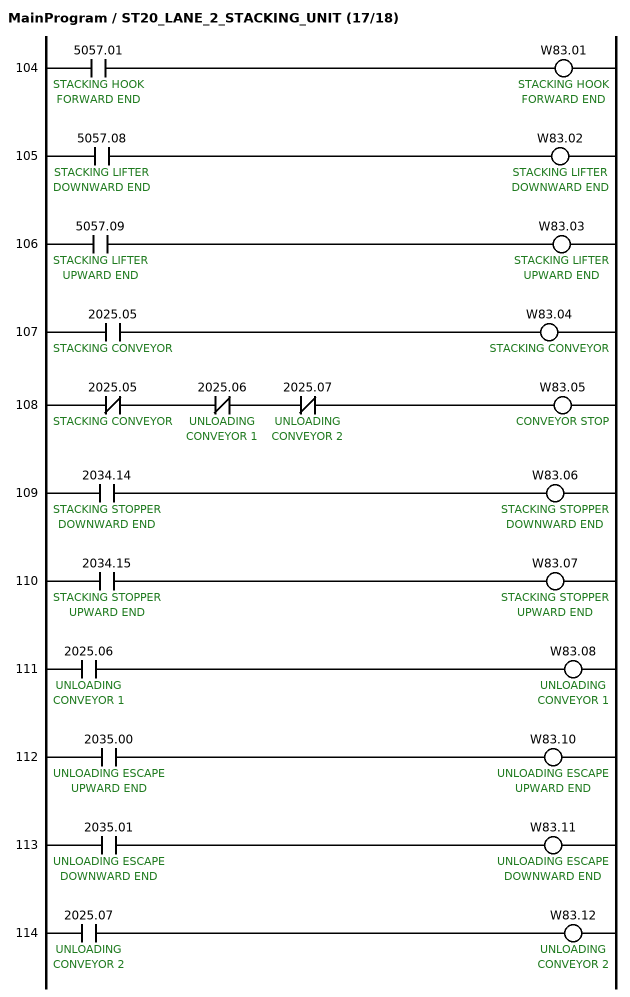
; [picture p720: MainProgram / ST20_LANE_2_STACKING_UNIT, rungs 104-114]
; rung 104
LD 5057.01  ; STACKING HOOK FORWARD END
OUT W83.01  ; STACKING HOOK FORWARD END
; rung 105
LD 5057.08  ; STACKING LIFTER DOWNWARD END
OUT W83.02  ; STACKING LIFTER DOWNWARD END
; rung 106
LD 5057.09  ; STACKING LIFTER UPWARD END
OUT W83.03  ; STACKING LIFTER UPWARD END
; rung 107
LD 2025.05  ; STACKING CONVEYOR
OUT W83.04  ; STACKING CONVEYOR
; rung 108
LDNOT 2025.05  ; STACKING CONVEYOR
ANDNOT 2025.06  ; UNLOADING CONVEYOR 1
ANDNOT 2025.07  ; UNLOADING CONVEYOR 2
OUT W83.05  ; CONVEYOR STOP
; rung 109
LD 2034.14  ; STACKING STOPPER DOWNWARD END
OUT W83.06  ; STACKING STOPPER DOWNWARD END
; rung 110
LD 2034.15  ; STACKING STOPPER UPWARD END
OUT W83.07  ; STACKING STOPPER UPWARD END
; rung 111
LD 2025.06  ; UNLOADING CONVEYOR 1
OUT W83.08  ; UNLOADING CONVEYOR 1
; rung 112
LD 2035.00  ; UNLOADING ESCAPE UPWARD END
OUT W83.10  ; UNLOADING ESCAPE UPWARD END
; rung 113
LD 2035.01  ; UNLOADING ESCAPE DOWNWARD END
OUT W83.11  ; UNLOADING ESCAPE DOWNWARD END
; rung 114
LD 2025.07  ; UNLOADING CONVEYOR 2
OUT W83.12  ; UNLOADING CONVEYOR 2

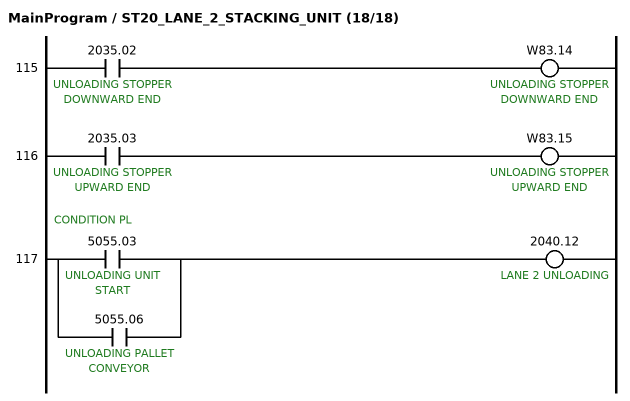
; rung 115
LD 2035.02  ; UNLOADING STOPPER DOWNWARD END
OUT W83.14  ; UNLOADING STOPPER DOWNWARD END
; rung 116
LD 2035.03  ; UNLOADING STOPPER UPWARD END
OUT W83.15  ; UNLOADING STOPPER UPWARD END
; rung 117: CONDITION PL
LD 5055.03  ; UNLOADING UNIT START
OR 5055.06  ; UNLOADING PALLET CONVEYOR
OUT 2040.12  ; LANE 2 UNLOADING

### Section End
; rung 0
END(001)